// TIA Portal V18 program export: 0 tag tables, 0 data types, 0 data blocks, 1 code blocks (in call order from the OBs), 0 instance data blocks

ORGANIZATION_BLOCK "Main"   // OB1, LAD, ProgramCycle
TITLE = "Main Program Sweep (Cycle)"
{ S7_Optimized_Access := 'TRUE' }
VERSION : 0.1
// stored: AutoNumber true, CodeModifiedDate 2021-05-25T13:42:20.5536351Z, CompileDate 2021-05-25T13:42:38.4564505Z, ConstantName OB_Main, CreationDate 2021-05-25T13:31:11.728453Z, EventClass Program cycle, HandleErrorsWithinBlock false, InterfaceModifiedDate 2008-07-21T16:55:08.419547Z, IsConsistent true, IsIECCheckEnabled false, IsKnowHowProtected false, IsWriteProtected false, ModifiedDate 2021-05-25T13:42:20.5536351Z, ParameterModified 2008-07-21T16:55:08.419547Z, PLCSimAdvancedSupport false, PriorityNumber 1, ProcessImagePartNumber 65535, SetENOAutomatically false, StructureModified 2008-07-21T16:55:08.419547Z
   VAR_INPUT
      Initial_Call : Bool;   // Initial call of this OB
      Remanence : Bool;   // =True, if remanent data are available
   END_VAR
BEGIN
END_ORGANIZATION_BLOCK
